ABB RobotStudio station: IRB2400 Palletizing.rsstn

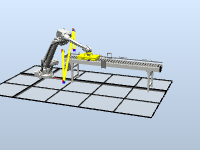
Station Solution2 (saved by RobotStudio 6.8.8148.134)
Controller System1
  mechanical unit ROB_1: IRB4600_20_250_C_01, 6 joints, base frame (0, 0, 0) mm
Layout (positions relative to the parent item):
  - 400_guide [part, from Equipment\Conveyor Guide 400.rslib] at (801.8, -220.36, 0) mm
  - IRB4600_20_250_C_01 [mechanism, from Robots\IRB4600_20_250_C_G_01.rslib] at (0, 0, 0) mm; joint values [-0.4475, 0.6481, -0.4427, 0, 1.3653, -6.7307] (rad or m)
  - tGripper [mechanism, from Libraries\tGripper.rslib] at (1871.95, -898.4, 1203.25) mm, rotated rx -180 ry 0 rz -180 deg
  - 工件 [part] at (3360.2, -20.14, 876.58) mm
  - 吸盘 [smart component]
      signals: DI di
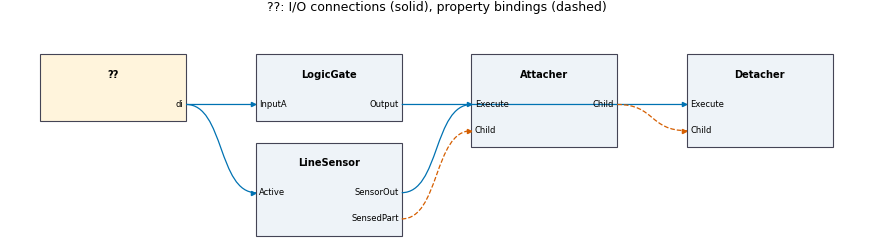
      connections:
        吸盘.di -> LogicGate.InputA
        LogicGate.Output -> Detacher.Execute
        吸盘.di -> LineSensor.Active
        LineSensor.SensorOut -> Attacher.Execute
        LineSensor.SensedPart => Attacher.Child
        Attacher.Child => Detacher.Child
    - LineSensor [smart component, from Components\LineSensor.rslib] at (1871.95, -898.4, 1043.25) mm, rotated rx -180 ry 0 rz -180 deg
        properties: Start=[-0.00999994765340695 3.46459762146767E-14 -0.00400000139453627]; End=[-0.00999995029097178 3.46459762146767E-14 0.0409999986054639]; Radius=0.05; SensedPart=(none); SensedPoint=[1.88194665527344 -0.898398742675781 0.296121704101563]
      - _sensorPart_ [part]
    - Attacher [smart component, from Components\Attacher.rslib]
        properties: Parent=tGripper; Flange=0; Child=(none); Mount=false; Offset=[0 0 0]; Orientation=[0 0 0]
    - Detacher [smart component, from Components\Detacher.rslib]
        properties: Child=(none); KeepPosition=true
    - LogicGate [smart component, from Components\LogicGate.rslib]
        properties: Operator=NOT; Delay=0
  - 传送带 [smart component]
      signals: DO do0
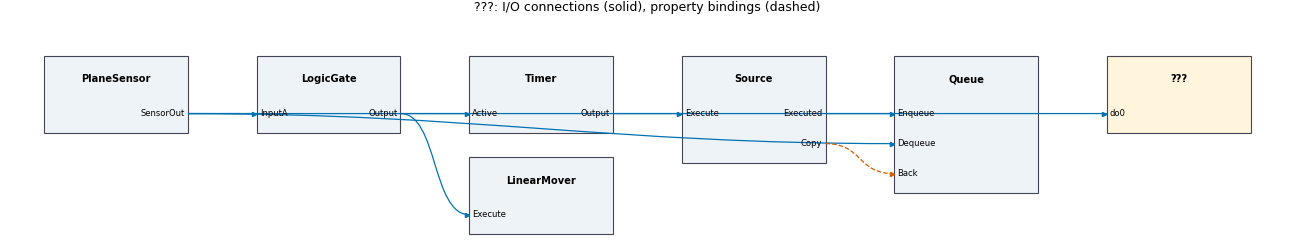
      connections:
        Timer.Output -> Source.Execute
        Source.Executed -> Queue.Enqueue
        PlaneSensor.SensorOut -> LogicGate.InputA
        LogicGate.Output -> LinearMover.Execute
        PlaneSensor.SensorOut -> Queue.Dequeue
        LogicGate.Output -> Timer.Active
        PlaneSensor.SensorOut -> 传送带.do0
        Source.Copy => Queue.Back
    - Timer [smart component, from Components\Timer.rslib]
        properties: StartTime=1; Interval=5; Repeat=true; CurrentTime=57.72
    - Source [smart component, from Components\Source.rslib]
        properties: Source=工件; Copy=(none); Parent=(none); Position=[3.360198 -0.02014 0.87658]; Orientation=[0 0 0]; Transient=false; PhysicsBehavior=0
    - Queue [smart component, from Components\Queue.rslib]
        properties: Back=(none); Front=(none); Queue={256844be-a364-4583-ae76-52d8d1d76155};{4fb5ce68-bf32-4061-af5b-054f3859f75d};{0eef695f-c43b-41b5-ab7a-de9741b1126a};{761b7318-9278-4e4c-902b-7f4ca79aecdd};{edafccec-ffed-4c27-a6f0-15b038c145a9};{e718deb0-e507-43f9-aedf-ff12c47128e1};{c19e9837-facb-4a8f-9fb0-2e5d1bbfb0c9};{59f9632f-e02f-4b81-a07f-684a1446da74};{01a5c4ce-8b5f-48aa-9084-c352b43b616f};{2eb9e72e-722c-466d-93b6-f4b7ae34aab6};{1ecdcdcc-0779-408b-a92e-08a26e1a40c1};{e07b5a67-2f57-4daa-ac93-0659555205b3};{ba36d030-219c-4bcf-a689-26d4a41c765f};{7e330409-6458-4764-967b-6aa65a062215};{0101a859-76b4-48e6-8f30-9077b41ecce5};{af5a4b1c-1827-4795-9622-ab6f452d8f69};{c7e296e4-9891-47be-aad9-a09093f8efc5};{856dbfec-1e97-41ba-bac1-18ae09a7c5b1};{49dde430-585b-4e08-b5cf-05bc97145806};{2134a6ce-5b60-453a-afcd-f51ebba49d7a};{f7d8f7d5-a887-4f17-afff-e800498add9c};{c08f6e4a-4274-40cd-97bc-bbbe92a4d0c7};{208c0b8e-ad24-4f82-8939-89d197414c24};{21f12e8b-bfa2-484f-89bb-23355336f71d};{9f47d88a-8342-4489-a5cd-7ef7728a0606};{8861541d-e5af-44af-8e48-bc64e7d55c75};{ebdf3481-8251-40e3-a234-c19c3dd71735};{e8665ef0-65ee-48b7-ba07-05a84002d8ca};{a9ae180b-1cc9-49a3-9eec-20de148f9d00};{e3291721-9c10-46df-9f4f-a7e3c6826097};{4cad2727-c97b-48a4-9865-657d64d1ae7a};{b0f1f9a0-0c07-4673-a19c-63c95a05b63f};{14c3c370-4796-45e3-9a7b-ee8a4075aae7};{f7470654-e6d5-414c-8c80-7484c4b0cc5e};{df76626a-9ea7-465f-9550-32c53e745612};{6ca7806c-98ee-4193-bb66-939fd42109c0};{bec20a0e-e92e-4180-810e-1b0e113e44e7};{27d798ce-9de0-43df-9b96-26b5f236c656};{77d466cb-fe0f-4b97-9d66-906481294d8b};{3784bb30-37fb-4e40-bc22-70bb66dd27d5};{df2b6f30-0e71-4696-85ce-c51d8b9b0f30};{c1b8587e-374d-49a6-87e3-3c0dc284dbd4};{796e77a8-4b57-4dd9-bac6-3454e177366f};{250e23be-7dc6-4f6d-9bdc-570fea1e1bd1};{d82ee078-1234-4034-b766-674d6af92af6};{3fb74582-b9a3-47ca-92c4-a811be5a83f8};{71f41479-5eb7-4a97-a5e1-d545e4ffc1c0};{48ad3dbe-e1f1-464a-99f9-b5a5218e4f4f};{a4ac2313-304e-44a9-96c2-5d5a9cb302bc};{d835151e-08bc-420f-9189-b641d70daa84};{62704fc7-2a43-4236-b215-c765123c4d58};{71a9cc92-652f-4c91-bd14-211720ef8c2a};{47bdfed7-637f-48a4-91db-90fb4607041d}; NumberOfObjects=2
    - PlaneSensor [smart component, from Components\PlaneSensor.rslib]
        properties: Origin=[0.821111 0.179642 0.77]; Axis1=[0 0 0.1]; Axis2=[0 -0.4 0]; SensedPart=(none)
      - _sensorPart_ [part]
    - LogicGate [smart component, from Components\LogicGate.rslib]
        properties: Operator=NOT; Delay=0
    - LinearMover [smart component, from Components\LinearMover.rslib]
        properties: Object=Queue; Direction=[-0.999 0 0]; Speed=0.2; Reference=Global; ReferenceObject=(none)
Attachment: tGripper is attached to IRB4600_20_250_C_01 / Link6
Attachment: LineSensor is attached to tGripper / tGripper
Station logic (signal -> signal, property => property):
  传送带.do0 -> System1.di00
  System1.do00 -> 吸盘.di
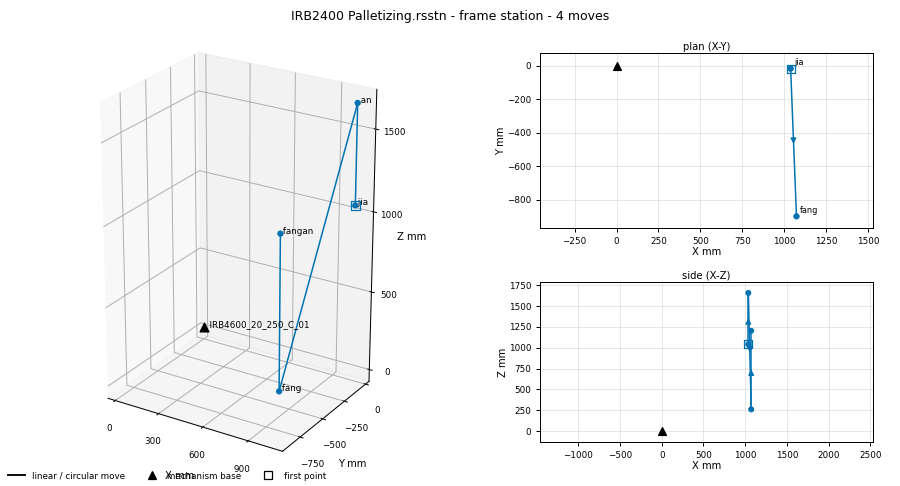
[picture p0: tool path of IRB2400 Palletizing.rsstn in frame station, 4 of 4 moves have a stored position in this frame; points joined in program order, loops and branches not executed]
Targets, tools, work objects and paths stored in the station, written as RAPID:
! task T_ROB1
MODULE CalibData
  PERS tooldata tGripper:=[TRUE,[[0,0,160],[1,0,0,0]],[1,[1,0,1],[1,0,0,0],0,0,0]];
ENDMODULE

! task T_ROB1
MODULE Module1
  CONST robtarget jia:=[[1037.144020762,-18.361904941,1041.9369747],[0.000004456,-0.000002927,1,-0.00000385],[-1,-1,-5,0],[9E+09,9E+09,9E+09,9E+09,9E+09,9E+09]];
  CONST robtarget an:=[[1037.143965988,-18.361909769,1656.980961796],[0.000004456,-0.000002964,1,-0.00000385],[-1,-1,-5,0],[9E+09,9E+09,9E+09,9E+09,9E+09,9E+09]];
  CONST robtarget fang:=[[1071.94514992,-898.397460373,261.479632626],[0.000004415,-0.000004467,1,-0.000003815],[-1,-1,-5,0],[9E+09,9E+09,9E+09,9E+09,9E+09,9E+09]];
  CONST robtarget fangan:=[[1071.946042003,-898.398230979,1203.253935617],[0.000004436,-0.000004474,1,-0.000003833],[-1,-1,-5,0],[9E+09,9E+09,9E+09,9E+09,9E+09,9E+09]];
  PROC Path_10()
    MoveL jia,v1000,z100,tool0\WObj:=wobj0;
    MoveL an,v1000,z100,tool0\WObj:=wobj0;
    MoveL fang,v1000,z100,tool0\WObj:=wobj0;
    MoveL fangan,v1000,z100,tool0\WObj:=wobj0;
  ENDPROC
ENDMODULE

